PROGRAM EnOceanSwitcher
VAR
	ftReceived: F_TRIG;
END_VAR

ftReceived(CLK:= EnOcean.bSwitchDataReceived, Q => received );
ftBtnBlue(CLK := GVL.btnBlue);

END_PROGRAM

(* stored: Version 1.1.0.1, ProductVersion 3.1.4024.11
   POU EnOceanSwitcher: Id {a0e4f2cf-8dbb-4098-9365-f32c54cbe2e4}, SpecialFunc None *)
